FUNCTION_BLOCK FB_WorkerDefGrid_Inspection EXTENDS FB_WorkerDefGrid
VAR_INPUT
  EL2252_Feedback      AT%I* : BYTE := 16#FF;   (*(optional from version > EL2252-0000-0018) Output feedback bit coded, needs activation in PDO config of terminal
                                              BIT 0: Output Kanal 1
                                              BIT 1: Tristate Kanal 1
                                              BIT 2: Output Kanal 2
                                              BIT 3: Tristate Kanal 2*)
  nCurrentPosition           : DINT;            // current position in [SubPx]
  fCurrentSpeed              : LREAL;           // current speed in [m/s]
  fMaxMachineSpeed           : LREAL;           // max. machine speed in [m/s]
END_VAR
VAR_OUTPUT
  // IOs
  EL2252_Activate      AT%Q* : BYTE;            (*Oututs activation command (0->3 activate)*)
  EL2252_StartTime     AT%Q* : T_DCTIME64;      (*Outputs activation timestamp*)
  EL2252_Output1       AT%Q* : BOOL;            (*Output1 bool state*)
END_VAR
VAR
  // timestamp output  
  tNowDc                          : T_DCTIME64;       // Get Current Timestamp (now)
  fCycleTime : LREAL;            // Current calculated cycle time [s]
  
  // helper
  nDistBtwTriggerAndInspection_SubPx : DINT;   // worker position in [SubPx]
  nTriggerPos_SubPx : DINT;   // next trigger position [SubPx]
  tTriggerTime : T_DCTIME64;
  bTriggerActivating, bOutputActive : BOOL;
  bTriggerResetting, bResetActive : BOOL;     // output is currently set
  tResetTime : T_DCTIME64;
  nDelta_SubPx : DINT;
END_VAR
VAR CONSTANT
  tC_CommTimeout : LREAL := 10.0/1000;   // 10ms in [s]
END_VAR

METHOD PROTECTED  Attach : BOOL
VAR_INPUT
  iCT              : I_CT;                         (*container at triggered event position*)
END_VAR
VAR
  // temp pos
  deltaPosNowToTrigger_SubPx : DINT;
  deltaPosNowToTrigger_m : LREAL;
  // temp time
  deltaTime_s : LREAL;
  deltaTime_Dc : T_DCTIME64;
END_VAR
IF SUPER^.Attach(iCT:=iCT) THEN
  
  // calculate exact trigger position
  // X0 + WorkerInspection-Pos
  nTriggerPos_SubPx := iCT.GetPosX0(iTracker:=_iCTTracker) + nDistBtwTriggerAndInspection_SubPx;
  // delta to current pos
  deltaPosNowToTrigger_SubPx := nTriggerPos_SubPx - nCurrentPosition;  // delata position in [SubPx]
  deltaPosNowToTrigger_m := F_SubPixelToMeter(lPosSubPx:=deltaPosNowToTrigger_SubPx, fResSubPx:=_fPrintResolution*_fSubPxResolution);
  
  IF fCurrentSpeed = 0 THEN RETURN; END_IF   // crash avoid
  // delta in time
  deltaTime_s  := deltaPosNowToTrigger_m/fCurrentSpeed;
  deltaTime_Dc := TO_ULINT(deltaTime_s * TO_LREAL(EC_DCTIME_TICKSPERSEC64));  
  
  // trigger time
  tTriggerTime := ULARGE_TO_ULINT(UInt64Add64(ULINT_TO_ULARGE(F_GetCurDcTaskTime64()), ULINT_TO_ULARGE(deltaTime_Dc)));
  setTrigger(bOut1:=TRUE, tTime:=tTriggerTime);
  bTriggerActivating := TRUE;
END_IF
END_METHOD

// cycle time in [s]
METHOD PRIVATE calcCycleTime : LREAL
VAR_INPUT
  tCurrent : T_DCTIME64;
END_VAR
VAR_INST
  tLastTimeStamp : T_DCTIME64 := 0;
END_VAR
calcCycleTime := (TO_LREAL(tCurrent) - TO_LREAL(tLastTimeStamp)) * 1E-9;
tLastTimeStamp  := tCurrent;  // memory timestamp
END_METHOD

METHOD   mJobStart
VAR_INPUT
	sJobDef	: I_JobDefinition;
END_VAR
END_METHOD

METHOD  mJobStop
VAR_INPUT
	sStatus	: I_JobStatus;
END_VAR
END_METHOD

METHOD Release : BOOL
VAR_INPUT
  iCT              : I_CT;                         (*container at triggered event position*)
END_VAR
IF SUPER^.Release(iCT := iCT) THEN
  ;  
END_IF
END_METHOD

METHOD PRIVATE resetOut
VAR
  tDistDc : T_DCTIME64;
  tULargeNow, tULargeDist : T_ULARGE_INTEGER;
END_VAR
// send FALSE in the next tC_CommTimeout
tDistDc := TO_ULINT(tC_CommTimeout * TO_LREAL(EC_DCTIME_TICKSPERSEC64));
tULargeNow := ULINT_TO_ULARGE(tNowDc);
tULargeDist := ULINT_TO_ULARGE(tDistDc);
tResetTime := ULARGE_TO_ULINT(UInt64Add64(tULargeNow, tULargeDist));
setTrigger(bOut1:=FALSE, tTime:=tResetTime);
END_METHOD

METHOD PRIVATE setTrigger
VAR_INPUT
  tTime : T_DCTIME64;
  bOut1 : BOOL;
END_VAR
EL2252_Activate  := 0;
EL2252_StartTime := tTime;
EL2252_Output1   := bOut1;
END_METHOD

METHOD  work
VAR
  bOutput1 : BOOL;
END_VAR
VAR_INST
  bTriggerActivating_mem : BOOL;
  bTriggerResetting_mem : BOOL;
  fPreAttachPos : LREAL;
END_VAR
SUPER^.work();

// Overwrite "default" tracking offset (Attach position)
fPreAttachPos := fMaxMachineSpeed * tC_CommTimeout;
_nTrackOffset := F_MeterToSubPixel(fPosMeter:=fPosition - fPreAttachPos, fResoSubPx:=_fPrintResolution*_fSubPxResolution);  // [pos domain] save position

// time & position updates
tNowDc     := F_GetCurDcTaskTime64();                         // current dc time (most accurate time stamp we have)
fCycleTime := calcCycleTime(tCurrent:=tNowDc);                // calculate cycle time of this fb
nDistBtwTriggerAndInspection_SubPx := F_MeterToSubPixel(fPosMeter:=fPosition, fResoSubPx:=_fPrintResolution*_fSubPxResolution);  // distance between Sensor and Inspectionin [SubPx] 

// output activation
IF bTriggerActivating AND bTriggerActivating_mem THEN  bTriggerActivating := FALSE;
  EL2252_Activate := 3;        // activate output config
  bOutputActive := TRUE;
END_IF
bTriggerActivating_mem := bTriggerActivating;

IF bOutputActive THEN
  // check if pos later than activation position --> reset
  nDelta_SubPx := F_MeterToSubPixel(fPosMeter:=tC_CommTimeout*fCurrentSpeed, fResoSubPx:=_fPrintResolution*_fSubPxResolution);
  IF (nCurrentPosition - nTriggerPos_SubPx) > nDelta_SubPx THEN
    resetOut();
    bTriggerResetting := TRUE;
    bOutputActive := FALSE;
	END_IF
END_IF

IF bTriggerResetting AND bTriggerResetting_mem THEN  bTriggerResetting := FALSE;
  EL2252_Activate := 3;        // activate output config
  bResetActive := TRUE;
END_IF
bTriggerResetting_mem := bTriggerResetting;

IF bResetActive THEN
  // check if pos later than activation position --> reset
  IF UInt64Cmp64(ULINT_TO_ULARGE(tNowDc), ULINT_TO_ULARGE(tResetTime)) > 0 THEN
    bResetActive := FALSE;
	END_IF
END_IF

IF _pAttachedCt <> 0 THEN
  Release(iCT:=_pAttachedCt^);
END_IF
END_METHOD

END_FUNCTION_BLOCK

(* stored: Version 1.1.0.1, ProductVersion 3.1.4024.11
   POU FB_WorkerDefGrid_Inspection: Id {d49e7280-4879-45fa-a34b-5703a36a2e59}, SpecialFunc None
   Folder EL2252: Id {0158c249-6857-46bf-a494-b2f1524d8491}
   Folder I_PrintStatusClient: Id {622e22de-7c75-455b-8827-a6bdaab0b713}
   Method Attach: Id {e841e17d-4c3c-4975-8ae0-07d1deff609f}
   Method calcCycleTime: Id {4f9d0544-5723-47c6-9b53-dcdf0a45a24d}
   Method mJobStart: Id {9e3e744c-c7cf-40e6-81f1-71a64963221a}
   Method mJobStop: Id {f410b542-746b-4eb1-9613-2986bd824a33}
   Method Release: Id {ecf27b47-fa13-4637-a110-5c617ebd743c}
   Method resetOut: Id {78afb77d-d3f3-44cd-9f32-46fd780b7dd5}
   Method setTrigger: Id {3e9e146e-8beb-4b75-a06e-084de4073f71}
   Method work: Id {c84e0ef9-4e1d-4b84-951f-24934b6f32d7} *)
